// TwinCAT 3 PLC project TestPLC
// ProgramVersion: 3.1.4023.0
// libraries:
//   Tc2_Standard, * (Beckhoff Automation GmbH)
//   Tc2_System, * (Beckhoff Automation GmbH)
//   Tc3_Module, * (Beckhoff Automation GmbH)
// project tree:
//   DUTs/ TestStruct.TcDUT (not stored), TestStruct2.TcDUT, TestStructComplex.TcDUT
//   GVLs/ GVL.TcGVL
//   / PlcTask.TcTTO (not stored)
//   POUs/ MAIN.TcPOU
// real-time tasks:
//   TASK PlcTask: cycle T#10ms, priority 20, ADS port 350

// ---- DUTs/TestStruct2.TcDUT
TYPE TestStruct2 :
STRUCT
	bTest			: BOOL := TRUE;
	fTestLreal		: LREAL := 77.777;
	sTest			: T_MAXSTRING := 'This could be a really long string...';
	//aInt			: ARRAY[0..2] OF INT;
END_STRUCT
END_TYPE

// ---- DUTs/TestStructComplex.TcDUT
TYPE TestStructComplex :
STRUCT
	iVal 	: DINT := 2;
	fVal 	: REAL := 2.2;
	sVal 	: STRING := 'Too many twos';
	stTest	: TestStruct2;
END_STRUCT
END_TYPE

// ---- GVLs/GVL.TcGVL
{attribute 'qualified_only'}
VAR_GLOBAL
	
	// PLC structure for testing type resolution in ADS client
	PlcStruct 			: TestStruct;
	PlcStructComplex	: TestStructComplex; // contains a struct inside this struct
	
	// Vars for client global event handler
	iEventData1 		: DINT := 1;
	fEventData2 		: REAL := 3.14;
	
	// Var for client custom event handler
	iCustomEvent 		: DINT := 2;
	
	// array for testing
	//aString				: ARRAY[0..4] OF STRING;
	
END_VAR

// ---- POUs/MAIN.TcPOU
PROGRAM MAIN
VAR
END_VAR

END_PROGRAM
